TYPE ST_SegmentIn :
STRUCT
END_STRUCT
END_TYPE

(* stored: Version 1.1.0.1
   DUT ST_SegmentIn: Id {d98fda91-c1c8-00f6-29f7-82f305f5b430} *)
